(* IEC 61131-3 sources: AutomationStudio/KomoraCieplna/OnOff, 3 files *)

(* ---- Types.typ ---- *)
TYPE
	cOnOffTyp : STRUCT
		Out : REAL; (* Zmienna sterująca CV - Output *)
		ActValue : REAL; (* Zmienna pomierzona PV - Input*)
		SetValue : REAL; (* Zmienna zadana SP - Input*)
		uiError : REAL; (* Błąd regulacji SP-PV - Calc*)
		Enable : BOOL; (* Aktywacja algorytmu - wysterowanie z poziomu KomCont*)
	END_STRUCT;
	cOnOffParTyp : STRUCT
		uiCVmax : REAL; (* Amplituda max sygnału CV *)
		uiCVmin : REAL; (* Ampliuda min sygnału CV *)
		uiEmax : REAL; (* Maksymalne odchylenie PV od SP *)
		uiEmin : REAL; (* Minimalne ochylenie PV od SP *)
		uiPVmax : REAL; (* Maksymalna wartość PV *)
		uiPVmin : REAL; (* Minimalna wartość PV *)
		uiLicznik : INT; (* Zmienna decydująca po ilu przejsciach proces może być w stanie ustalonym *)
		uiAutoTuningOnOff : BOOL:=TRUE; (* Zmienna włączająca lub wyłączająca auto strojenie *)
	END_STRUCT;

	AutoTuningTyp : STRUCT
		fTempOnOff : BOOL; (* flaga do wyznaczenia wykresuy PU *)
		flag : BOOL:=FALSE; (* flaga do sprawdzenia czy przy edgepos wystartować, czy zakończyc zegar *)
		P : REAL; (* zmienna mierząca okres *)
		Amplituda : REAL; (* Zmienna przechowująca Amax-Amin *)
		Amax : REAL; (* Zmienna przechowująca maksymalne odchylenie aplitudy  *)
		Amin : REAL; (* Zmienna przechowująca minimalne odchylenie aplitudy  *)
		K : REAL; (* Zmienna K wyliczona ze wzoru *)
		fLicznik : INT; (* Licznik, który kontroluje przejscie procesu w stan ustalony *)
		H : REAL;
	END_STRUCT;

END_TYPE

(* ---- Main.st ---- *)
PROGRAM _INIT
	AutoTuning.Amax:=gKomoraPar[0].TemperatureSP;
	AutoTuning.Amin:=gKomoraPar[0].TemperatureSP;
END_PROGRAM

PROGRAM _CYCLIC
	//AutoTuning.Amin:=gKomoraPar[0].TemperatureSP;
	cOnOff[0].ActValue:= gOnOff.TemperaturePV; (* Pobranie wartości temperatury w KomCont *)
	gOnOff.HeaterCV:= cOnOff[0].Out; (* Wysłanie sygnału sterującego grzałką do KomCont *)
	gAutoTuningOnOff:=cOnOffPar[0].uiAutoTuningOnOff;
	cOnOff[0].SetValue:= gKomoraPar[0].TemperatureSP; (* Pobranie wartości zadanej z GUI *)
	cOnOff[0].Enable:= gOnOff.Enable; (* Aktywacja będzie z poziomu KomCont Start-Stop*)
	cOnOff[0].uiError:= cOnOff[0].SetValue - cOnOff[0].ActValue; (* SP-PV -> węzeł sumacyjny -> Schemat *)

	IF EDGEPOS(cOnOff[0].Enable) THEN 					(* Przystosowanie parametrów do startu algorytmu *)
		AutoTuning.flag:=FALSE;  						(* flaga do startu/stopu zegarka *)
		AutoTuning.P:=0;								(* Zmienna przechowywująca okres od CVpos do CVpos *)
		AutoTuning.Amax:=gKomoraPar[0].TemperatureSP;   (* Przypisanie wartości Max (ponieważ program mógł być wcześniej uruchomiony - i mogła zostać tam poprzednia wartość ) *)
		AutoTuning.Amin:=gKomoraPar[0].TemperatureSP;	(* Przypisanie wartości Min (ponieważ program mógł być wcześniej uruchomiony - i mogła zostać tam poprzednia wartość ) *)
	END_IF;

	IF cOnOff[0].Enable = TRUE THEN
		IF cOnOff[0].uiError >= cOnOffPar[0].uiEmax THEN
			cOnOff[0].Out:= cOnOffPar[0].uiCVmax;
			AutoTuning.fTempOnOff:=TRUE;				(* flaga wskazująca czy CV uległo zmianie *)
		ELSIF cOnOff[0].uiError <= cOnOffPar[0].uiEmin THEN
			cOnOff[0].Out:= cOnOffPar[0].uiCVmin;
			AutoTuning.fTempOnOff:=FALSE;				(* flaga wskazująca czy CV uległo zmianie *)
		END_IF;
	ELSE
		cOnOff[0].Out:= 0; (* Zatrzymanie procesu sterowania - wciśnięcie Stop bądź E-Stop *)
	END_IF;

	(* Główna część eksperymentu przekaźnikowego *)
	IF (cOnOff[0].Enable AND cOnOffPar[0].uiAutoTuningOnOff) AND (AutoTuning.fLicznik >cOnOffPar[0].uiLicznik) THEN (* Licznik po to aby sprawdzić czy proces jest w stanie quasi-stabilnym *)
		(* Szukanie max i min amplitudy *)
		IF gOnOff.TemperaturePV>AutoTuning.Amax THEN
			AutoTuning.Amax:=gOnOff.TemperaturePV;
		ELSIF gOnOff.TemperaturePV<AutoTuning.Amin THEN
			AutoTuning.Amin:=gOnOff.TemperaturePV;
		END_IF;

		(* Odmierzenie okresu od załączonego CV do załączonego CV *)
		IF EDGEPOS(AutoTuning.fTempOnOff) THEN
			AutoTuning.flag:=NOT(AutoTuning.flag);
			DelayTON[1].IN:=AutoTuning.flag;
			DelayTON[1].PT:=T#1h;
			IF AutoTuning.flag=FALSE THEN
	 			 AutoTuning.P:=(TIME_TO_REAL(DelayTON[1].ET)/1000);
			END_IF;
		END_IF;
	END_IF;

	IF EDGENEG(AutoTuning.fTempOnOff) AND cOnOffPar[0].uiAutoTuningOnOff THEN (* Dodawanie do licznika (wartość SP+Emin przekroczona) *)
		AutoTuning.fLicznik:=AutoTuning.fLicznik+1;
	END_IF;

	(* Wyliczenie wartości Kp,Ti,Td oraz przekazanie ich do globalnych zmiennych *)
	IF EDGENEG(cOnOff[0].Enable) AND cOnOffPar[0].uiAutoTuningOnOff THEN
		AutoTuning.H:=(cOnOffPar[0].uiCVmax-cOnOffPar[0].uiCVmin)/2;
		AutoTuning.Amplituda:=(AutoTuning.Amax-AutoTuning.Amin)/2;
		AutoTuning.K:=(4*AutoTuning.H)/(3.14159265359*AutoTuning.Amplituda);
		gKp:=0.6*AutoTuning.K;
		gTi:=AutoTuning.P/2;
		gTd:=AutoTuning.P/8;
		AutoTuning.fLicznik:=0;		(* Przygotowanie zmiennych do ponownego uruchomienia *)
		AutoTuning.flag:=FALSE;
	END_IF;

	DelayTON[1]();
END_PROGRAM

PROGRAM _EXIT
	(* Insert code here *)

END_PROGRAM

(* ---- Variables.var ---- *)
VAR
	cOnOff : ARRAY[0..1] OF cOnOffTyp; (* Struktura algorytmu OnOff *)
	DelayTON : ARRAY[0..10] OF TON; (* zegarki *)
	LiczMinMax : ARRAY[0..10] OF LCRMinMax; (* Funkcja liczenia min i max *)
	AutoTuning : AutoTuningTyp;

END_VAR

VAR RETAIN
	cOnOffPar : ARRAY[0..1] OF cOnOffParTyp; (* Struktura parametrów algorytmu OnOff *)

END_VAR
